FUNCTION_BLOCK FB_DiagnosisEtherCATSlaveWc1
VAR_OUTPUT
	bError						:BOOL;								//エラー発生を出力
END_VAR
VAR
	_eEtherCATSlave				:E_EtherCATSlave;
	
	fbStateDiagnosis			:FB_StateDiagnosis;
	fbWcStateDiagnosis			:FB_WcStateDiagnosis;
END_VAR

//診断用FBを呼び出し
fbStateDiagnosis(eEtherCATSlave:=_eEtherCATSlave);
fbWcStateDiagnosis(eEtherCATSlave:=_eEtherCATSlave);

bError:=fbStateDiagnosis.bError OR fbWcStateDiagnosis.bError;

//FB_Init は常に暗黙的に使用可能で、主に初期化に使用されます。
//戻り値は評価されません。特定の結果を得るために、メソッドを明示的に宣言し、
//そのメソッドに標準の初期化コードをもったコードを追加することができます。戻り値を評価できます。
METHOD FB_Init: BOOL
VAR_INPUT
    bInitRetains: BOOL; // TRUE: 保持変数は初期化されます (ウォーム リセット、あるいはコールド リセット)
    bInCopyCode: BOOL;  // TRUE: 後でコードをコピーする (オンライン変更) ために、インスタンスをコピーします。

	eEtherCATSlave							:E_EtherCATSlave;
END_VAR
_eEtherCATSlave:=eEtherCATSlave;
END_METHOD

END_FUNCTION_BLOCK

(* stored: Version 1.1.0.1, ProductVersion 3.1.4026.18
   POU FB_DiagnosisEtherCATSlaveWc1: Id {e5af8d40-9ba8-4884-bbf0-fd8f1590eb8a}, SpecialFunc None
   Method FB_Init: Id {968a1203-d202-47ce-a297-b0203464f442} *)
